FUNCTION_BLOCK AI_GENERATED_ADD_INT
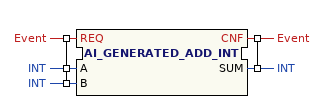
  EVENT_INPUT
    REQ WITH A, B;
  END_EVENT
  EVENT_OUTPUT
    CNF WITH SUM;
  END_EVENT
  VAR_INPUT
    A : INT;
    B : INT;
  END_VAR
  VAR_OUTPUT
    SUM : INT;
  END_VAR
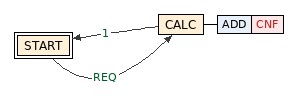
  EC_STATES
    START;
    CALC : ADD -> CNF;
  END_STATES
  EC_TRANSITIONS
    START TO CALC := REQ;
    CALC TO START := 1;
  END_TRANSITIONS
  ALGORITHM ADD IN ST:
SUM := A + B;
  END_ALGORITHM
END_FUNCTION_BLOCK
